// TIA Portal V16 export
// export: Created 2021-11-12T13:31:53.3850307Z, ExportSetting WithDefaults, DisplayName Totally Integrated Automation Portal, DisplayVersion V16 Update 3, DisplayName TIA Portal Version Control Interface, DisplayVersion V16 Update 2, DisplayName TIA Portal Openness, DisplayVersion V16 Update 3, DisplayName SINAMICS Startdrive Advanced, DisplayVersion V16 Update 5, DisplayName SINAMICS Startdrive G130, G150, S120, S150, SINAMICS MV, S210, DisplayVersion V16 Update 5, DisplayName SINAMICS Startdrive G110M, G120, G120C, G120D, G120P, G115D, DisplayVersion V16 Update 5, DisplayName STEP 7 Professional, DisplayVersion V16 Update 3, DisplayName STEP 7 Safety, DisplayVersion V16, DisplayName WinCC UA Professional, DisplayVersion V16 Update 3
DATA_BLOCK "IDB_Cab_000+UH10"   // DB64
VERSION : 0.1
// stored: AutoNumber true, DBAccessibleFromOPCUA true, InstanceOfName Cab_000+UH10, InstanceOfType FB
"Cab_000+UH10"
   // VAR
   //    SF_EC01_3_Alarm { S7_SetPoint := 'True'} : "STD_DI_Mon";
   //    SF_FC21_14_Alarm { S7_SetPoint := 'True'} : "STD_DI_Mon";
   //    SF_FC22_14_Alarm { S7_SetPoint := 'True'} : "STD_DI_Mon";
   //    SF_FB02_14_Alarm { S7_SetPoint := 'True'} : "STD_DI_Mon";
   //    SF_SF22_14_Alarm { S7_SetPoint := 'True'} : "STD_DI_Mon";
   // END_VAR
BEGIN
END_DATA_BLOCK
